PROGRAM main
  VAR
    START_PB AT %IX0.0 : BOOL;
    STOP_PB AT %IX0.1 : BOOL;
    E_STOP AT %IX0.2 : BOOL;
    ENTRY_SEN AT %IX0.3 : BOOL;
    VISION_REJECT_FLAG AT %QX0.3 : BOOL;
    VISION_HEARTBEAT AT %QX0.4 : BOOL;
    EXIT_SEN AT %IX0.6 : BOOL;
    CONV_MOTOR_1 AT %QX0.0 : BOOL;
    CONV_MOTOR_2 AT %QX0.5 : BOOL;
    CONV_MOTOR_3 AT %QX0.6 : BOOL;
    REJECT_SOL AT %QX0.1 : BOOL;
    FAULT_LAMP AT %QX0.2 : BOOL;
    OBJ_PRESENT : BOOL;
    TON0 : TON;
    HB_PULSE : BOOL;
    R_TRIG0 : R_TRIG;
    TOF0 : TOF;
    TOF1 : TOF;
  END_VAR

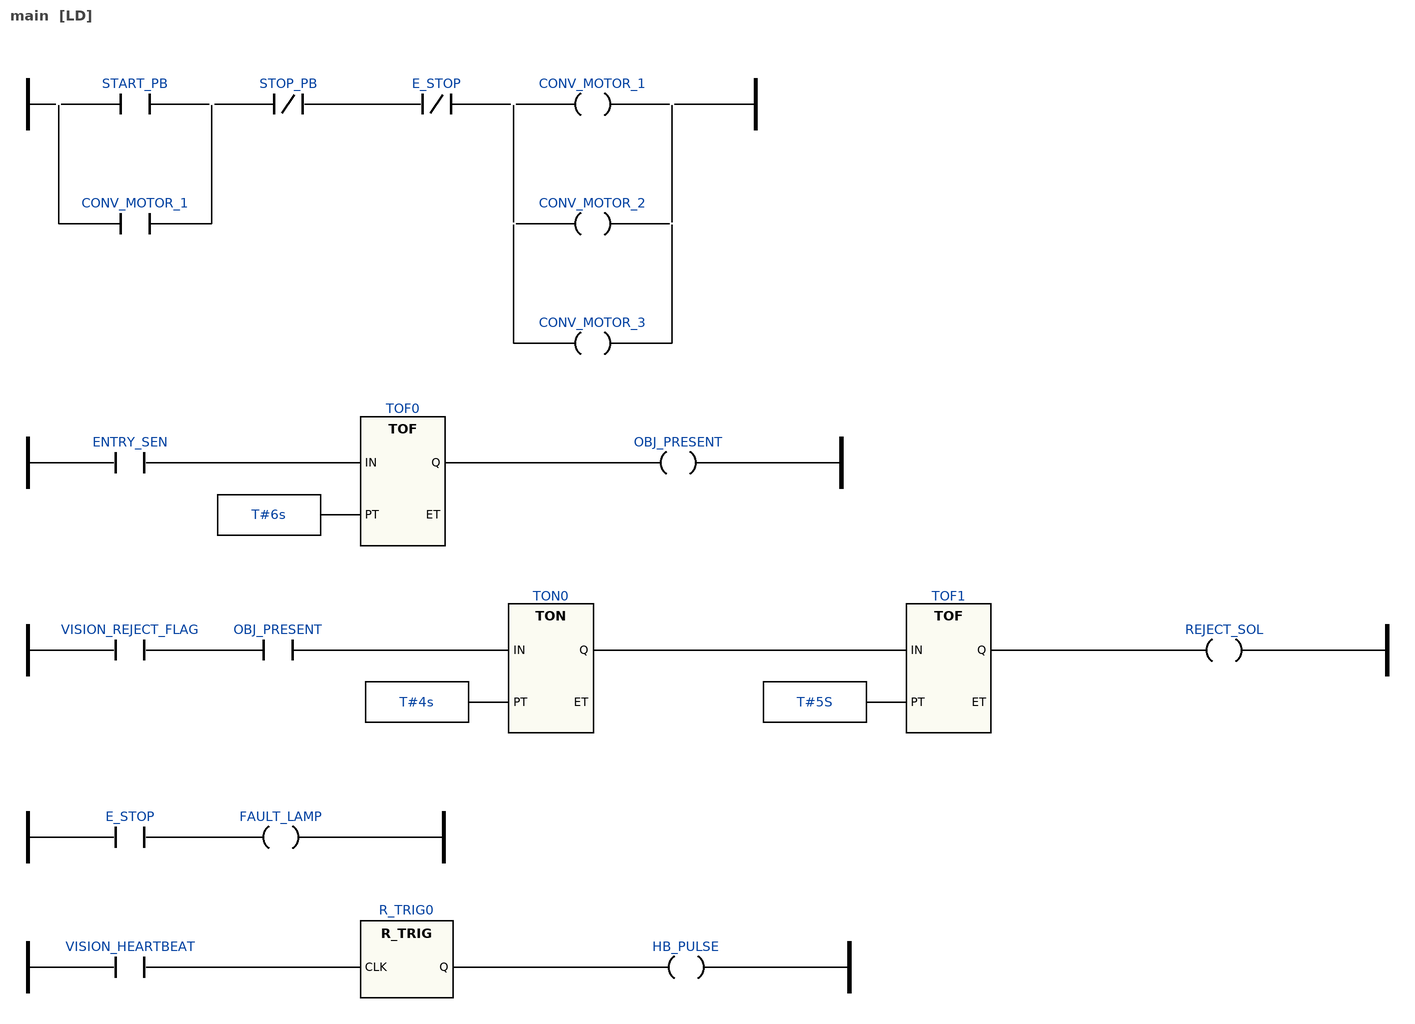
(* LD diagram, written out as Structured Text *)
CONV_MOTOR_1 := (START_PB OR CONV_MOTOR_1) AND NOT STOP_PB AND NOT E_STOP;
CONV_MOTOR_2 := (START_PB OR CONV_MOTOR_1) AND NOT STOP_PB AND NOT E_STOP;
CONV_MOTOR_3 := (START_PB OR CONV_MOTOR_1) AND NOT STOP_PB AND NOT E_STOP;
TOF0(IN := ENTRY_SEN, PT := T#6s);
OBJ_PRESENT := TOF0.Q;
TON0(IN := VISION_REJECT_FLAG AND OBJ_PRESENT, PT := T#4s);
TOF1(IN := TON0.Q, PT := T#5S);
REJECT_SOL := TOF1.Q;
FAULT_LAMP := E_STOP;
R_TRIG0(CLK := VISION_HEARTBEAT);
HB_PULSE := R_TRIG0.Q;
END_PROGRAM
